FUNCTION_BLOCK FB_SequenceHelperSb EXTENDS FB_SequenceHelper
VAR_INPUT
END_VAR
VAR_OUTPUT
END_VAR
VAR
	wsb 			: FB_WStringBuilder;
	iInfoTextId		: INT;
	wsInfoTextId 	: WSTRING;
END_VAR

SUPER^();

PROPERTY PUBLIC Info : REFERENCE TO FB_WStringBuilder
GET
Info Ref= wsb;
END_GET
END_PROPERTY

PROPERTY PUBLIC InfoTextId : INT
GET
InfoTextId := iInfoTextId;
END_GET
SET
iInfoTextId := InfoTextId;
END_SET
END_PROPERTY

PROPERTY PUBLIC InfoTextWsId : WSTRING
GET
InfoTextWsId := wsInfoTextId;
END_GET
SET
wsInfoTextId := InfoTextWsId;
END_SET
END_PROPERTY

METHOD PUBLIC SetInfo : BOOL
VAR_INPUT
	stInfo : ST_Text;
END_VAR
iInfoTextId := stInfo.nNameId;
wsb.Set(stInfo.wsName);
wsInfoTextId := stInfo.wsNameId;
END_METHOD

END_FUNCTION_BLOCK

(* stored: Version 1.1.0.1
   POU FB_SequenceHelperSb: Id {bcf99656-7ad2-47fc-ab2f-9b2be02aa13f}, SpecialFunc None
   Property Info: Id {80474ce1-b87d-45cf-ae1b-7abdf012e9cc}
   Get Get: Id {2c3277fa-3d3a-446a-84ff-b48029e89c47}
   Property InfoTextId: Id {01dde9df-d404-4259-a18d-c2a1fa1e90c5}
   Get Get: Id {f01b7fdf-d428-48a4-9122-398f04159b2f}
   Set Set: Id {13989555-d239-4255-95f1-4e75b7e7fbce}
   Property InfoTextWsId: Id {770ab5c3-87a9-40ff-bbce-8d0e717e1d3e}
   Get Get: Id {0d26ca09-6c9a-4987-8fea-9bc334b78dd3}
   Set Set: Id {4e185fe0-8c86-4614-ac94-247f598961c4}
   Method SetInfo: Id {3047607d-e78c-4a31-8dc5-0a4a1b0ce1db} *)
